{attribute addProperty BoxType "EK1122-0000-0018"}
{attribute addProperty Id "Beckhoff_ELM31xxsub_EK1100EK1100_179A0949162"}
{attribute addProperty CRC "1041719436"}
{attribute addProperty SizeInBites "16"}
{attribute addProperty SizeInBytes "2"}
TYPE Beckhoff_ELM31xxEK1122_3E17608C EXTENDS EK1122_179A0949 :
STRUCT
	{attribute addProperty Name "Beckhoff_ELM31xxsub_EK1100"}
	Beckhoff_ELM31xxsub_EK1100 : EK1100_179A0949;
END_STRUCT
END_TYPE

(* stored: Version 1.2.0.0, ProductVersion 3.1.4024.9
   DUT Beckhoff_ELM31xxEK1122_3E17608C: Id {334cce8d-48ac-40c1-b343-2c87f4774aee} *)
